FUNCTION_BLOCK FB_N2_DEVICE
VAR_INPUT
	AlarmConfig : TYP_ALARM_DEVICE_CONFIG;
END_VAR
VAR_OUTPUT
END_VAR
VAR
	bTestalarm : BOOL;
	bTestReset : BOOL;
	bTestAcknowledge : BOOL;
	fbPurgeN2DeviceError : FB_ALARM;
END_VAR

fbPurgeN2DeviceError.Config.Acknowledge := E_ALARM_ACK_TYPE.ACK_AND_RESET;
fbPurgeN2DeviceError.Config.Name := CONCAT(AlarmConfig.Name, '*PURGE_N2_GENERAL_ERROR');
fbPurgeN2DeviceError.Config.Priority := 3;
fbPurgeN2DeviceError(Handler := AlarmConfig.Handler);

IF bTestalarm THEN
	fbPurgeN2DeviceError.Activate();
ELSIF bTestReset THEN
	fbPurgeN2DeviceError.Reset();
ELSIF bTestAcknowledge THEN
	fbPurgeN2DeviceError.Acknowledge();
END_IF

END_FUNCTION_BLOCK

(* stored: Version 1.1.0.1, ProductVersion 3.1.4024.12
   POU FB_N2_DEVICE: Id {f0b43921-35fb-4e47-b654-653011a067a3}, SpecialFunc None *)
